TYPE TupleStruct_1:
    STRUCT
        field0: LREAL;
        field1: LREAL;
        field2: LREAL;
        field3: LREAL;
        field4: LREAL;
        field5: LREAL;
        field6: LREAL;
        field7: LREAL;
        field8: LREAL;
        field9: LREAL;
        field10: LREAL;
        field11: LREAL;
        field12: LREAL;
        field13: LREAL;
    END_STRUCT
END_TYPE

(* stored: ProductVersion 3.1.0.18, Version 1.1.0.1 *)
